
// ===== library: MasterCopy "lineer_calculater" =====

FUNCTION_BLOCK "lineer_calculater"   // FB1, LAD
{ S7_Optimized_Access := 'TRUE' }
VERSION : 0.1
   VAR_INPUT
      X : Real;
      X1 : Real;
      X0 : Real;
      Y1 : Real;
      Y0 : Real;
   END_VAR
   VAR_OUTPUT
      Y : Real;
   END_VAR
BEGIN

REGION Network 1
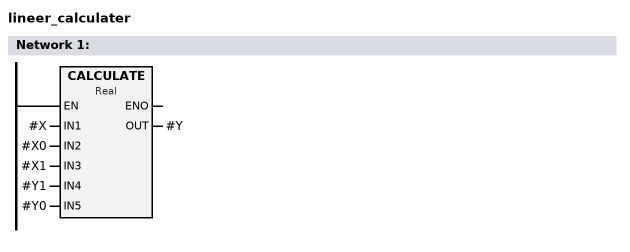
   RUNG wire#powerrail
      { S7_Templates := "SrcType := Real"; S7_Expression := "((IN4-IN5)/(IN3-IN2)*(IN1-IN2))+IN5" } Calculate(in1 := #X, in2 := #X0, in3 := #X1, in4 := #Y1, in5 := #Y0, out => #Y)
   END_RUNG
   // the same network as SCL:
   #Y := ((#Y1-#Y0)/(#X1-#X0)*(#X-#X0))+#Y0;
END_REGION
END_FUNCTION_BLOCK